{attribute 'GeneratedUsingTerminal: EJ2522-0000-0022'}
{attribute addProperty BoxType "EJ2522-0000-0022"}
{attribute addProperty Id "Set_counterBOOL1ReservedBOOL1"}
{attribute addProperty CRC "2833108354"}
{attribute addProperty Size "2"}
TYPE Control_A8DDCD82 :
STRUCT
	{attribute addProperty Name "Set_counter"}
	Set_counter : BOOL;
	{attribute addProperty Name "Reserved"}
	Reserved : BOOL;
END_STRUCT
END_TYPE

(* stored: Version 1.2.0.0, ProductVersion 3.1.4024.9
   DUT Control_A8DDCD82: Id {ddfbcae3-884b-4262-9fe5-f1f2d3d0627f} *)
